{attribute 'GeneratedUsingTerminal: KL9999'}
{attribute addProperty BoxType "KL9999"}
{attribute addProperty Id "VarInAT %I*UINT0VarOutAT %Q*UINT0"}
{attribute addProperty CRC "308619075"}
{attribute addProperty Size "0"}
TYPE Channel_12652743 :
STRUCT
	{attribute addProperty Name "VarIn"}
	VarIn AT %I* : UINT;
	{attribute addProperty Name "VarOut"}
	VarOut AT %Q* : UINT;
END_STRUCT
END_TYPE

(* stored: Version 1.2.0.0, ProductVersion 3.1.4024.9
   DUT Channel_12652743: Id {eebe4eae-a4d8-4143-af27-6853be922f56} *)
